FUNCTION fMembershipDegree : real
VAR_INPUT
	CrispInput: REAL;
	MF:MEMBERSHIP_FUNCTION;
END_VAR

VAR_OUTPUT
	error: BOOL;
END_VAR

CASE MF.Shape OF
	MF_SHAPE.Gaussian://********
		fMembershipDegree:=
			MF_Gaussian(
				x:= CrispInput,
				c:= MF.Points[1],
				d:= MF.Points[2],
				Error=>error);
	MF_SHAPE.Lshaped://********
		fMembershipDegree:=
			MF_L(
				x:= CrispInput,
				a:= MF.Points[1],
				b:= MF.Points[2],
				Error=>error);

	MF_SHAPE.rshaped://********
		fMembershipDegree:=
			MF_R(
				x:= CrispInput,
				c:= MF.Points[1],
				d:= MF.Points[2],
				Error=>error);
	
	MF_SHAPE.Sshaped://********
		fMembershipDegree:=
			MF_S(
				x:= CrispInput,
				a:= MF.Points[1],
				b:= MF.Points[2],
				Error=>error);

	MF_SHAPE.Sigmoidal://********
		fMembershipDegree:=
			MF_Gaussian(
				x:= CrispInput,
				d:= MF.Points[1],
				c:= MF.Points[2],
				Error=>error);
							
	MF_SHAPE.Singleton://********
		fMembershipDegree:=
			MF_Singleton(
				x:= CrispInput,
				a:= MF.Points[1]);
				
	MF_SHAPE.Trapeziodal://********
		fMembershipDegree:=
			MF_Trapezoidal(
				x:= CrispInput,
				a:= MF.Points[1],
				b:= MF.Points[2],
				c:= MF.Points[3],
				d:= MF.Points[3],
				Error=>error);
	
	MF_SHAPE.Triangular://********	
		fMembershipDegree:=
			MF_Triangular(
				x:= CrispInput,
				a:= MF.Points[1],
				m:= MF.Points[2],
				b:= MF.Points[3],
				error=>error);
				
	MF_SHAPE.Zshaped://********
		fMembershipDegree:=
			MF_R(
				x:= CrispInput,
				c:= MF.Points[1],
				d:= MF.Points[2],
				Error=>error);
	ELSE
		error:=TRUE;
	END_CASE;

END_FUNCTION

(* stored: Version 1.1.0.1, ProductVersion 3.1.4024.6
   POU fMembershipDegree: Id {5864e0d4-c664-4471-9579-ecccf008b753}, SpecialFunc None *)
